SUBAPPLICATION Uebung_003f_AX (* DigitalInput_I1-8 auf DigitalOutput_Q1-8 *)
  (* Standard: 61499-2; Description: Copyright (c) 2026 Meisterschulen am Ostbahnhof This program and the accompanying materials are made available under the terms of the Eclipse Public License 2.0 which is available at https://www.eclipse.org/legal/epl-2.0/ SPDX-License-Identifier: EPL-2.0 *)
  (* Version 1.0, 2026-10-05, Franz Höpfinger, Meisterschulen am Ostbahnhof, initial API and implementation and/or initial documentation - wie Uebung_003b_AX, aber alle 8 Kanaele statt nur 4 *)
  PACKAGE Uebungen;
  IMPORT logiBUS::io::DI::logiBUS_DI::Input_I1;
  IMPORT logiBUS::io::DI::logiBUS_DI::Input_I2;
  IMPORT logiBUS::io::DI::logiBUS_DI::Input_I3;
  IMPORT logiBUS::io::DI::logiBUS_DI::Input_I4;
  IMPORT logiBUS::io::DI::logiBUS_DI::Input_I5;
  IMPORT logiBUS::io::DI::logiBUS_DI::Input_I6;
  IMPORT logiBUS::io::DI::logiBUS_DI::Input_I7;
  IMPORT logiBUS::io::DI::logiBUS_DI::Input_I8;
  IMPORT logiBUS::io::DQ::logiBUS_DO::Output_Q1;
  IMPORT logiBUS::io::DQ::logiBUS_DO::Output_Q2;
  IMPORT logiBUS::io::DQ::logiBUS_DO::Output_Q3;
  IMPORT logiBUS::io::DQ::logiBUS_DO::Output_Q4;
  IMPORT logiBUS::io::DQ::logiBUS_DO::Output_Q5;
  IMPORT logiBUS::io::DQ::logiBUS_DO::Output_Q6;
  IMPORT logiBUS::io::DQ::logiBUS_DO::Output_Q7;
  IMPORT logiBUS::io::DQ::logiBUS_DO::Output_Q8;
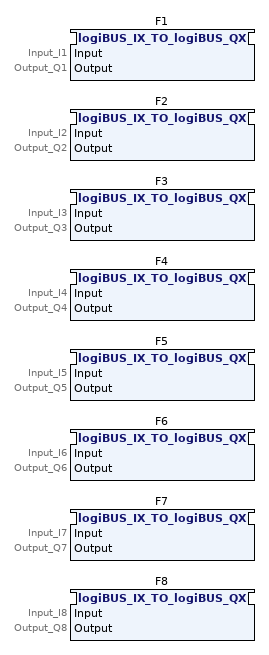
  SUBAPPS
    F1 : MyLib::sys::logiBUS_IX_TO_logiBUS_QX(Input := Input_I1, Output := Output_Q1);
    F2 : MyLib::sys::logiBUS_IX_TO_logiBUS_QX(Input := Input_I2, Output := Output_Q2);
    F3 : MyLib::sys::logiBUS_IX_TO_logiBUS_QX(Input := Input_I3, Output := Output_Q3);
    F4 : MyLib::sys::logiBUS_IX_TO_logiBUS_QX(Input := Input_I4, Output := Output_Q4);
    F5 : MyLib::sys::logiBUS_IX_TO_logiBUS_QX(Input := Input_I5, Output := Output_Q5);
    F6 : MyLib::sys::logiBUS_IX_TO_logiBUS_QX(Input := Input_I6, Output := Output_Q6);
    F7 : MyLib::sys::logiBUS_IX_TO_logiBUS_QX(Input := Input_I7, Output := Output_Q7);
    F8 : MyLib::sys::logiBUS_IX_TO_logiBUS_QX(Input := Input_I8, Output := Output_Q8);
  END_SUBAPPS
END_SUBAPPLICATION
